(* PLC project canopen_master, beremiz beremiz 1 *)
(* stored: creationDateTime 2008-06-24T18:44:00, modificationDateTime 2009-10-07T18:45:11, language en-US *)

PROGRAM test_main
  VAR
    PLC_OUT AT %QW0.0.2.8193.0 : INT;
    PLC_IN AT %IW0.0.2.8192.0 : INT;
  END_VAR

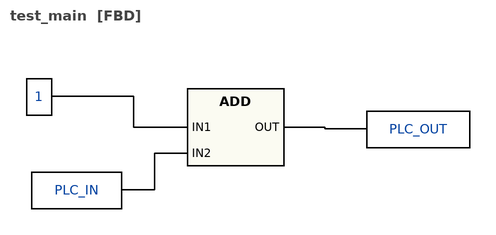
(* FBD diagram, written out as Structured Text *)
PLC_OUT := 1 + PLC_IN;
END_PROGRAM

CONFIGURATION conf
  RESOURCE res ON PLC
    TASK tache(INTERVAL := t#50ms, PRIORITY := 0);
    PROGRAM toto WITH tache : test_main;
  END_RESOURCE
END_CONFIGURATION
